INTERFACE I_Objekt_SmartGreifer

METHOD M_Reset : BOOL
VAR_INPUT
END_VAR
END_METHOD

METHOD M_Start : BOOL
VAR_INPUT
END_VAR
END_METHOD

METHOD M_Stop : BOOL
VAR_INPUT
END_VAR
END_METHOD

PROPERTY P_Prozessparameter : sSmartGreiferProzessVariablen
SET
END_SET
END_PROPERTY

PROPERTY P_State : eObjectState
GET
END_GET
END_PROPERTY

END_INTERFACE

(* stored: Version 1.1.0.1
   Itf I_Objekt_SmartGreifer: Id {1623e398-1fd1-40e2-bd39-c723e9818eb6}
   Method M_Reset: Id {8dc2480f-3d49-4c19-9178-1b5e43fe339a}
   Method M_Start: Id {f55f07b2-8b98-433b-98de-f19ab19679e3}
   Method M_Stop: Id {cc9f4680-6034-4211-b89c-e0c4b6520672}
   Property P_Prozessparameter: Id {85a5ded3-c2ce-4155-b393-bcbd5a05c330}
   Set Set: Id {9b63eca7-3408-4517-ab17-1d51f31c9292}
   Property P_State: Id {f4e0b349-8551-4263-85d3-47d7fe655d20}
   Get Get: Id {1a87ea74-f84d-43c6-8e6b-fa808289347a} *)
